(* IEC 61131-3 sources: plc_generation_empirical_study/our_method_delta_DVP48ES300R/calibration/timer_scan_semantics, 1 file *)

(* ---- candidate.st ---- *)
FUNCTION_BLOCK DVP_TimerScanCalibration
VAR_INPUT
    Enable : BOOL;
END_VAR
VAR_OUTPUT
    CounterDone : BOOL;
    TimerDone : BOOL;
END_VAR
VAR
    ScanCount : INT := 0;
    DelayTimer : TON;
END_VAR

IF NOT Enable THEN
    ScanCount := 0;
ELSIF ScanCount < 4 THEN
    ScanCount := ScanCount + 1;
END_IF;

DelayTimer(IN := Enable, PT := T#300ms);
CounterDone := ScanCount >= 4;
TimerDone := DelayTimer.Q;
END_FUNCTION_BLOCK
